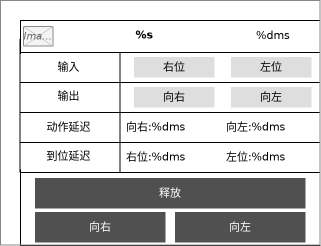
VISUALIZATION Cylinder4  // 321x246
VAR_INPUT
	System:							REFERENCE TO ST_System;
	Cylinder:						REFERENCE TO ST_Cylinder;
	CylinderData:					REFERENCE TO ST_CylinderData;
END_VAR
    RoundedRectangle (20,131 300x115)
    RoundedRectangle (20,20 300x115)
    Rectangle (20,54 300x115)
    Line (20,52) (320,52)
    Rectangle (55,23 179x24), "%s", text variable: Cylinder.arrInfo[System.stMode.eLanguage].sName, input disabled if: Cylinder.stLock.bShield
    Rectangle (238,23 70x25), "%dms", text variable: CylinderData.iAlarmTime, input disabled if: Cylinder.stLock.bShield
        OnMouseClick: write the text variable via VisuDialogs.Numpad
    Line (20,82) (320,82)
    Line (20,112) (320,112)
    Label (21,52 95x30), "输入"
    Label (21,81 95x30), "输出"
    Line (120,172) (120,52)
    RoundedRectangle (134,57 80x20), "右位", colour toggle: Cylinder.stInput.bWork, input disabled if: Cylinder.stLock.bShield
    RoundedRectangle (231,57 80x20), "左位", colour toggle: Cylinder.stInput.bHome, input disabled if: Cylinder.stLock.bShield
    RoundedRectangle (134,87 80x20), "向右", colour toggle: Cylinder.stOutput.bWork, input disabled if: Cylinder.stLock.bShield
    RoundedRectangle (231,87 80x20), "向左", colour toggle: Cylinder.stOutput.bHome, input disabled if: Cylinder.stLock.bShield
    RoundedRectangle (35,178 270x30), "释放", colour toggle: Cylinder.stLock.bOff OR Cylinder.stLock.bAll, input disabled if: Cylinder.stLock.bShield
        tap Cylinder.stControl.stOffRequest.bManual
    RoundedRectangle (35,212 130x30), "向右", colour toggle: Cylinder.stLock.bWork OR Cylinder.stLock.bAll, input disabled if: Cylinder.stLock.bShield
        tap Cylinder.stControl.stWorkRequest.bManual
    RoundedRectangle (175,212 130x30), "向左", colour toggle: Cylinder.stLock.bHome OR Cylinder.stLock.bAll, input disabled if: Cylinder.stLock.bShield
        tap Cylinder.stControl.stHomeRequest.bManual
    Line (320,174) (320,43)
    Line (20,172) (20,39)
    Image (23,26 30x20), image: ImagePool.Cylinder1
    Line (20,142) (320,142)
    Line (20,172) (320,172)
    Label (21,112 95x30), "动作延迟"
    Label (21,141 95x30), "到位延迟"
    RoundedRectangle (123,114 95x26), "向右:%dms", text variable: CylinderData.iWorkRequestTime, input disabled if: Cylinder.stLock.bShield
        OnMouseClick: write the text variable via Default
    RoundedRectangle (223,114 95x26), "向左:%dms", text variable: CylinderData.iHomeRequestTime, input disabled if: Cylinder.stLock.bShield
        OnMouseClick: write the text variable via Default
    RoundedRectangle (123,144 95x26), "右位:%dms", text variable: CylinderData.iWorkDone, input disabled if: Cylinder.stLock.bShield
        OnMouseClick: write the text variable via Default
    RoundedRectangle (223,144 95x26), "左位:%dms", text variable: CylinderData.iHomeDone, input disabled if: Cylinder.stLock.bShield
        OnMouseClick: write the text variable via Default
END_VISUALIZATION

(* stored: Version 1.1.0.1, ProductVersion 3.1.4024.4
   Visu Cylinder4: Id {916e6fe6-24b6-41b9-84b7-eb0938afa1f7} *)
